FUNCTION_BLOCK ABSTRACT FB_DigitalOutputBase IMPLEMENTS I_DigitalOutput
VAR
	_overrideEnable : BOOL;
	_overrideValue : BOOL;
	_rawInput : BOOL;
	_value : BOOL;
END_VAR

PROPERTY OverrideEnable : BOOL
GET
OverrideEnable := _overrideEnable;
END_GET
SET
_overrideEnable := OverrideEnable;
END_SET
END_PROPERTY

PROPERTY OverrideValue : BOOL
GET
OverrideValue := _overrideValue;
END_GET
SET
_overrideValue := OverrideValue;
END_SET
END_PROPERTY

PROPERTY RawInput : BOOL
GET
RawInput := _rawInput;
END_GET
SET
_rawInput := RawInput;
END_SET
END_PROPERTY

METHOD Run
IF _overrideEnable THEN
	_value := _overrideValue;
ELSE
	_value := _rawInput;
END_IF
END_METHOD

PROPERTY Value : BOOL
GET
Value := _value;
END_GET
END_PROPERTY

END_FUNCTION_BLOCK

(* stored: Version 1.1.0.1, ProductVersion 3.1.4026.18
   POU FB_DigitalOutputBase: Id {20d7a993-bee3-49fb-a834-6412ab94a790}, SpecialFunc None
   Property OverrideEnable: Id {47d7ff60-e835-4f24-975a-c1728a6c7565}
   Get Get: Id {9e525c42-3365-4cc7-848c-1fbacc999da6}
   Set Set: Id {dad7c668-56e3-4ba8-ad2c-6729c655d09e}
   Property OverrideValue: Id {3e5ac6a1-ab7f-4a45-8130-47526d7cb274}
   Get Get: Id {4033c320-2d45-4758-9d78-55f77c4c4330}
   Set Set: Id {76cd7468-46ce-42ac-a872-84d89107a034}
   Property RawInput: Id {3b5b7fca-61b9-4a8a-8fbf-07a2bc89b051}
   Get Get: Id {6d06faaa-18c3-4eb9-958f-ff78a136148d}
   Set Set: Id {98bdcbce-0178-434b-a268-70f2a329920a}
   Method Run: Id {22c6521e-5bdf-44e1-8546-00727e9f2686}
   Property Value: Id {7dc50187-5a46-4612-9ae0-7828c177469d}
   Get Get: Id {0f9b262d-4157-45c6-8d9a-eeca4e750c4e} *)
